// TIA Portal V19 export
FUNCTION "AnalogWriteValues" : Void   // FC9, STL
TITLE = Write Analog Output Value
{ S7_Optimized_Access := 'TRUE' }
VERSION : 0.0
// Comment
// stored: AutoNumber false
   VAR_TEMP
      scratch_int : Int;
   END_VAR
BEGIN

NETWORK
TITLE = Write Analog Output Value, IP01.49/50
      CALL  "AnalogWritingSystem"
      ( OUT_VAL     := "STP_PT0167/IP0149_50".IP0149OutSTP,
        MIN_REAL    := 0.0,
        MAX_REAL    := 10000.0,
        OUT_DA_CONV := "P_IP014950":P
      );


NETWORK
TITLE = Write Analog Output Value, IP01.57
      CALL  "AnalogWritingSystem"
      ( OUT_VAL     := "PID_TT0172/IP0157".IP0157OuPID,
        MIN_REAL    := 0.0,
        MAX_REAL    := 10000.0,
        OUT_DA_CONV := "P_IP0157":P
      );


NETWORK
TITLE = Re-transmit Analog Input Value, WT01.69
      L     "P_WT0169":P;
      T     #scratch_int;

      CALL  "AnalogWritingSystem"
      ( OUT_VAL     := #scratch_int,
        MIN_REAL    := 0.0,
        MAX_REAL    := 15000.0,
        OUT_DA_CONV := "P_WT0169_TX":P
      );

END_FUNCTION
